FUNCTION_BLOCK FloorSensors (* Composite Function Block Type *)
  (* Standard: 61499-2 *)
  (* Version 0.0, 7/12/2016, Andrei, nxtControl GmbH, template *)
  PACKAGE Main;
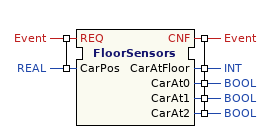
  EVENT_INPUT
    REQ WITH CarPos; (* Normal Execution Request *)
  END_EVENT
  EVENT_OUTPUT
    CNF WITH CarAtFloor, CarAt0, CarAt1, CarAt2; (* Execution Confirmation *)
  END_EVENT
  VAR_INPUT
    CarPos : REAL; (* Input event qualifier *)
  END_VAR
  VAR_OUTPUT
    CarAtFloor : INT; (* Output event qualifier *)
    CarAt0 : BOOL;
    CarAt1 : BOOL;
    CarAt2 : BOOL;
  END_VAR
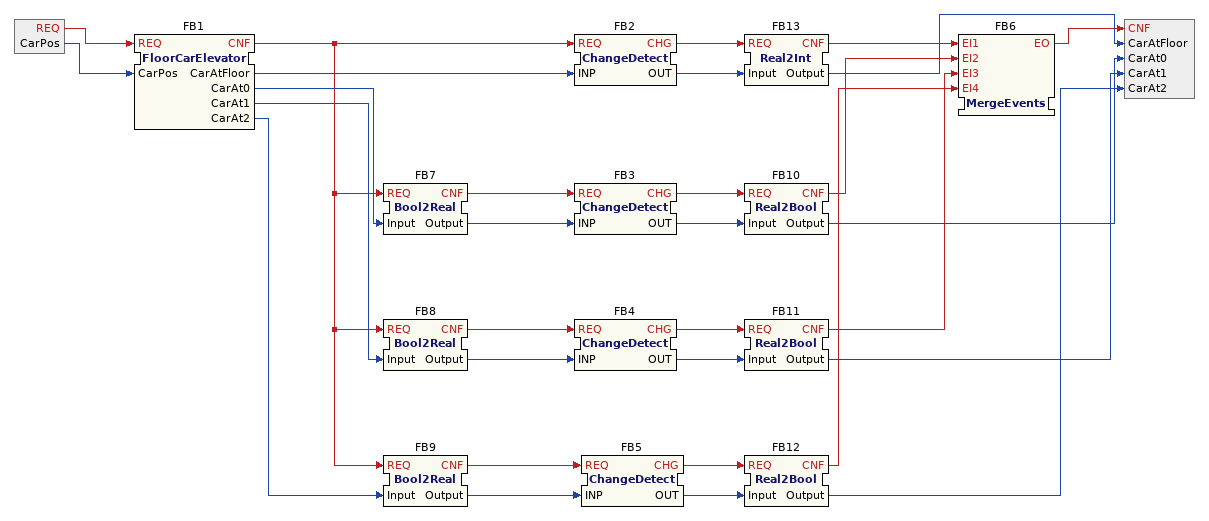
  FBS
    FB1 : FloorCarElevator;
    FB2 : ChangeDetect;
    FB3 : ChangeDetect;
    FB4 : ChangeDetect;
    FB5 : ChangeDetect;
    FB6 : MergeEvents;
    FB7 : Bool2Real;
    FB8 : Bool2Real;
    FB9 : Bool2Real;
    FB10 : Real2Bool;
    FB11 : Real2Bool;
    FB12 : Real2Bool;
    FB13 : Real2Int;
  END_FBS
  EVENT_CONNECTIONS
    FB1.CNF TO FB2.REQ;
    FB1.CNF TO FB7.REQ;
    FB1.CNF TO FB8.REQ;
    FB1.CNF TO FB9.REQ;
    FB2.CHG TO FB13.REQ;
    FB3.CHG TO FB10.REQ;
    FB4.CHG TO FB11.REQ;
    FB5.CHG TO FB12.REQ;
    REQ TO FB1.REQ;
    FB6.EO TO CNF;
    FB7.CNF TO FB3.REQ;
    FB8.CNF TO FB4.REQ;
    FB9.CNF TO FB5.REQ;
    FB10.CNF TO FB6.EI2;
    FB11.CNF TO FB6.EI3;
    FB12.CNF TO FB6.EI4;
    FB13.CNF TO FB6.EI1;
  END_CONNECTIONS
  DATA_CONNECTIONS
    FB1.CarAtFloor TO FB2.INP;
    FB1.CarAt0 TO FB7.Input;
    FB1.CarAt1 TO FB8.Input;
    FB1.CarAt2 TO FB9.Input;
    FB4.OUT TO FB11.Input;
    FB5.OUT TO FB12.Input;
    FB3.OUT TO FB10.Input;
    FB2.OUT TO FB13.Input;
    CarPos TO FB1.CarPos;
    FB7.Output TO FB3.INP;
    FB8.Output TO FB4.INP;
    FB9.Output TO FB5.INP;
    FB10.Output TO CarAt0;
    FB11.Output TO CarAt1;
    FB12.Output TO CarAt2;
    FB13.Output TO CarAtFloor;
  END_CONNECTIONS
END_FUNCTION_BLOCK
